// SIMATIC S7-200 project (STEP 7-Micro/WIN), CPU 224XP REL 02.01

ORGANIZATION_BLOCK MAIN:OB1
TITLE=PROGRAM COMMENTS
BEGIN
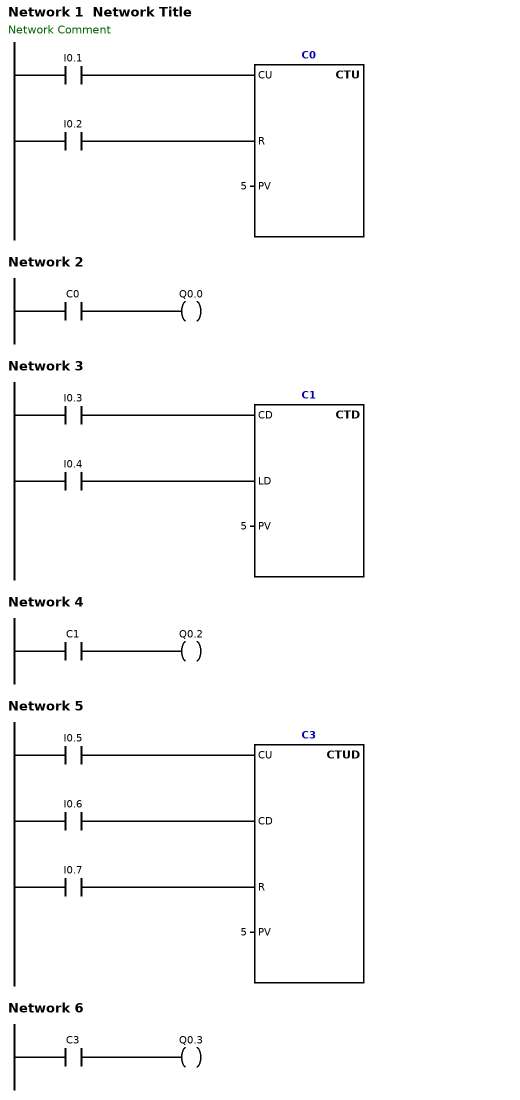
Network 1 // Network Title
// Network Comment
LD     I0.1
LD     I0.2
CTU    C0, 5
Network 2
LD     C0
=      Q0.0
Network 3
LD     I0.3
LD     I0.4
CTD    C1, 5
Network 4
LD     C1
=      Q0.2
Network 5
LD     I0.5
LD     I0.6
LD     I0.7
CTUD   C3, 5
Network 6
LD     C3
=      Q0.3
END_ORGANIZATION_BLOCK
